// TIA Portal V17 export
// export: Created 2025-03-07T09:18:55.9761065Z, ExportSetting WithDefaults, DisplayName Totally Integrated Automation Portal, DisplayVersion V17 Update 8, DisplayName TIA Portal Openness, DisplayVersion V17 Update 8, DisplayName TIA Portal Version Control Interface, DisplayVersion V17, DisplayName SINAMICS Startdrive Advanced, DisplayVersion V17 SP2, DisplayName SINAMICS Startdrive G110M, G120, G120C, G120D, G120P, G115D, DisplayVersion V17 SP2, DisplayName SINAMICS Startdrive G130, G150, S120, S150, SINAMICS MV, S210, DisplayVersion V17 SP2, DisplayName STEP 7 Professional, DisplayVersion V17 Update 8, DisplayName SINUMERIK ONE STEP 7 Toolbox, DisplayVersion V17 Update 12, DisplayName SINUMERIK 840D sl STEP 7 Toolbox, DisplayVersion V17 Update 12, DisplayName STEP 7 Safety, DisplayVersion V17 Update 6, DisplayName WinCC Advanced, DisplayVersion V17 Update 8
FUNCTION "FC20300_TARGET_LIGHT_COORDINATOR" : Void   // FC20300, LAD
TITLE = FC20300 TARGET LIGHT COORDINATOR
{ S7_Optimized_Access := 'TRUE' }
VERSION : 0.1
// stored: AutoNumber false, IsIECCheckEnabled false, SetENOAutomatically false, UDAEnableTagReadback false
BEGIN

REGION Network 1: CALL FB20300 LASER GUIDE UNIT 1
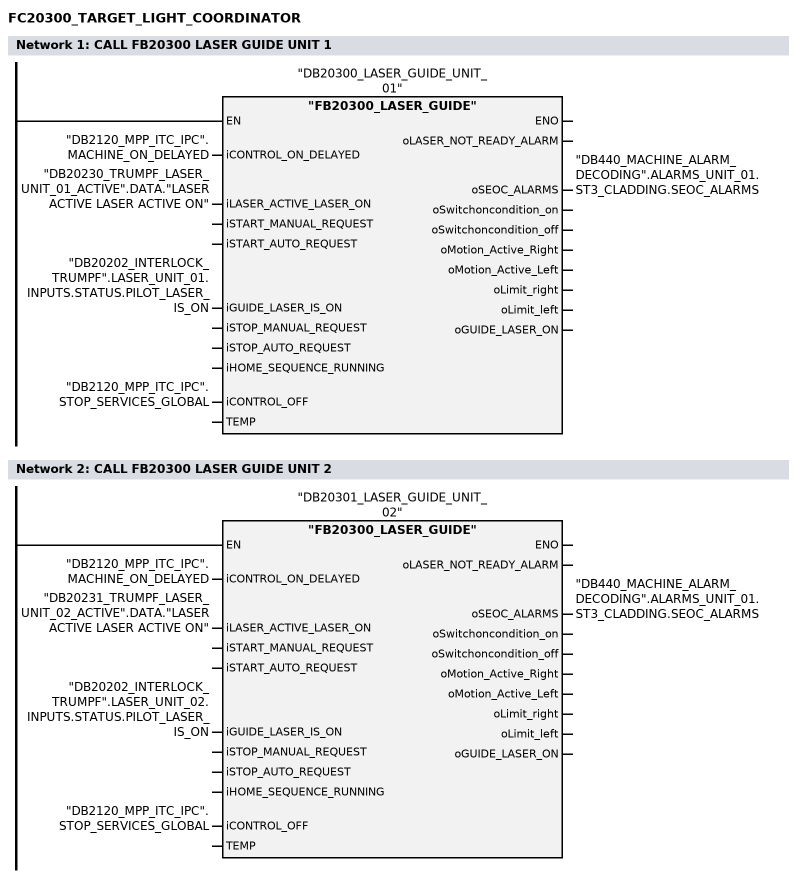
   RUNG wire#powerrail
      "DB20300_LASER_GUIDE_UNIT_01"(iCONTROL_ON_DELAYED := "DB2120_MPP_ITC_IPC".MACHINE_ON_DELAYED, iLASER_ACTIVE_LASER_ON := "DB20230_TRUMPF_LASER_UNIT_01_ACTIVE".DATA."LASER ACTIVE LASER ACTIVE ON", iSTART_MANUAL_REQUEST :=, iSTART_AUTO_REQUEST :=, iGUIDE_LASER_IS_ON := "DB20202_INTERLOCK_TRUMPF".LASER_UNIT_01.INPUTS.STATUS.PILOT_LASER_IS_ON, iSTOP_MANUAL_REQUEST :=, iSTOP_AUTO_REQUEST :=, iHOME_SEQUENCE_RUNNING :=, iCONTROL_OFF := "DB2120_MPP_ITC_IPC".STOP_SERVICES_GLOBAL, TEMP :=, oLASER_NOT_READY_ALARM =>, oSEOC_ALARMS => "DB440_MACHINE_ALARM_DECODING".ALARMS_UNIT_01.ST3_CLADDING.SEOC_ALARMS, oSwitchoncondition_on =>, oSwitchoncondition_off =>, oMotion_Active_Right =>, oMotion_Active_Left =>, oLimit_right =>, oLimit_left =>, oGUIDE_LASER_ON =>)
   END_RUNG
   // the same network as SCL:
   "DB20300_LASER_GUIDE_UNIT_01"(iCONTROL_ON_DELAYED := "DB2120_MPP_ITC_IPC".MACHINE_ON_DELAYED,   // "FB20300_LASER_GUIDE"
                           iLASER_ACTIVE_LASER_ON := "DB20230_TRUMPF_LASER_UNIT_01_ACTIVE".DATA."LASER ACTIVE LASER ACTIVE ON",
                           iGUIDE_LASER_IS_ON := "DB20202_INTERLOCK_TRUMPF".LASER_UNIT_01.INPUTS.STATUS.PILOT_LASER_IS_ON,
                           iCONTROL_OFF := "DB2120_MPP_ITC_IPC".STOP_SERVICES_GLOBAL,
                           oSEOC_ALARMS => "DB440_MACHINE_ALARM_DECODING".ALARMS_UNIT_01.ST3_CLADDING.SEOC_ALARMS);
END_REGION

REGION Network 2: CALL FB20300 LASER GUIDE UNIT 2
   RUNG wire#powerrail
      "DB20301_LASER_GUIDE_UNIT_02"(iCONTROL_ON_DELAYED := "DB2120_MPP_ITC_IPC".MACHINE_ON_DELAYED, iLASER_ACTIVE_LASER_ON := "DB20231_TRUMPF_LASER_UNIT_02_ACTIVE".DATA."LASER ACTIVE LASER ACTIVE ON", iSTART_MANUAL_REQUEST :=, iSTART_AUTO_REQUEST :=, iGUIDE_LASER_IS_ON := "DB20202_INTERLOCK_TRUMPF".LASER_UNIT_02.INPUTS.STATUS.PILOT_LASER_IS_ON, iSTOP_MANUAL_REQUEST :=, iSTOP_AUTO_REQUEST :=, iHOME_SEQUENCE_RUNNING :=, iCONTROL_OFF := "DB2120_MPP_ITC_IPC".STOP_SERVICES_GLOBAL, TEMP :=, oLASER_NOT_READY_ALARM =>, oSEOC_ALARMS => "DB440_MACHINE_ALARM_DECODING".ALARMS_UNIT_01.ST3_CLADDING.SEOC_ALARMS, oSwitchoncondition_on =>, oSwitchoncondition_off =>, oMotion_Active_Right =>, oMotion_Active_Left =>, oLimit_right =>, oLimit_left =>, oGUIDE_LASER_ON =>)
   END_RUNG
   // the same network as SCL:
   "DB20301_LASER_GUIDE_UNIT_02"(iCONTROL_ON_DELAYED := "DB2120_MPP_ITC_IPC".MACHINE_ON_DELAYED,   // "FB20300_LASER_GUIDE"
                           iLASER_ACTIVE_LASER_ON := "DB20231_TRUMPF_LASER_UNIT_02_ACTIVE".DATA."LASER ACTIVE LASER ACTIVE ON",
                           iGUIDE_LASER_IS_ON := "DB20202_INTERLOCK_TRUMPF".LASER_UNIT_02.INPUTS.STATUS.PILOT_LASER_IS_ON,
                           iCONTROL_OFF := "DB2120_MPP_ITC_IPC".STOP_SERVICES_GLOBAL,
                           oSEOC_ALARMS => "DB440_MACHINE_ALARM_DECODING".ALARMS_UNIT_01.ST3_CLADDING.SEOC_ALARMS);
END_REGION
END_FUNCTION
